{attribute 'linkalways'} 
{attribute 'no_explicit_call' := 'This FB is a CLASS and must be accessed using methods or properties'}
{attribute 'enable_dynamic_creation'}
FUNCTION_BLOCK Node_F_VN_ContourRoundness EXTENDS VisionNode
VAR
    ipContour : _ITcVnContainer;
    fRoundness : _LREAL(0.0);
    hrPrev : _HRESULT(S_OK);
	hresult : _HRESULT(S_OK);
END_VAR

METHOD PUBLIC  Clone : I_Node
VAR
	pNode : POINTER TO Node_F_VN_ContourRoundness;
END_VAR
pNode := __NEW(Node_F_VN_ContourRoundness);
Clone := pNode^;
END_METHOD

METHOD FB_init : BOOL
VAR_INPUT
	bInitRetains : BOOL; // if TRUE, the retain variables are initialized (warm start / cold start)
	bInCopyCode : BOOL;  // if TRUE, the instance afterwards gets moved into the copy code (online change)
END_VAR
AddInput('ipContour', ipContour);
AddInput('hrPrev', hrPrev);
AddOutput('fRoundness', fRoundness);
AddOutput('hresult',hresult);
END_METHOD

METHOD PROTECTED OnExecute
hresult.Value := F_VN_ContourRoundness(
	ipContour := ipContour.Value,
    fRoundness := fRoundness.Value,
	hrPrev:= hrPrev.Value);
END_METHOD

METHOD PUBLIC PreExecutionCheck
VAR_INPUT
	Check : I_PreExecutionChecks;
END_VAR
Check.IsTrue(ipContour.IsValid, 'ipContour must be a valid container');
Check.IsTrue((ipContour.IsType(TC_GLOBAL_CONST_LIST.ContainerType_Vector_TcVnPoint2_DINT) OR
              ipContour.IsType(TC_GLOBAL_CONST_LIST.ContainerType_Vector_TcVnPoint2_REAL)),
              'ipContour contains incorrect type');
END_METHOD

END_FUNCTION_BLOCK

(* stored: Version 1.1.0.1, ProductVersion 3.1.4026.13
   POU Node_F_VN_ContourRoundness: Id {a74ed07a-2f22-09f5-0cb0-2d513b91ffd8}, SpecialFunc None
   Folder Constructor: Id {f5dcebbd-a42f-0dd0-168d-96b08b1d78e6}
   Method Clone: Id {05388173-e1d0-057f-1f4a-fcd803e184b0}
   Method FB_init: Id {dad51b9f-cb1b-0e8e-0f09-2e50d40acdfb}
   Method OnExecute: Id {d4a94b2b-bd45-08db-2fe0-e4b6964ccbbc}
   Method PreExecutionCheck: Id {05f3f27b-662b-0846-2f3c-0aa231e731d7} *)
